(*

## Short summary
An interface to provide configurations for cycle manager steps.
Used internally to allow better fluent implementation.

.. <legal notes>

legal notes
=================
| SPDX-FileCopyrightText: © 2024 ekvip automation GmbH <info@ekvip.de>
| SPDX-License-Identifier: Apache-2.0
| For details check: Apache-2.0_

.. _Apache-2.0: https://www.apache.org/licenses/LICENSE-2.0

.. </legal notes>



*)
INTERFACE INTERNAL ICycleManagerStepParameters EXTENDS __System.IQueryInterface

PROPERTY currentErrorStep : DINT
SET
END_SET
END_PROPERTY

PROPERTY currentPauseEnabled : BOOL
SET
END_SET
END_PROPERTY

PROPERTY currentSteppingEnabled : BOOL
SET
END_SET
END_PROPERTY

PROPERTY currentStepWidth : DINT
SET
END_SET
END_PROPERTY

PROPERTY currentStopRequestMode :CNM_CycleManagerInterfaces.StepStopRequestMode
SET
END_SET
END_PROPERTY

PROPERTY currentTimeout : TIME
SET
END_SET
END_PROPERTY

PROPERTY currentTimeoutStep : DINT
SET
END_SET
END_PROPERTY

END_INTERFACE

(* stored: Version 1.1.0.1
   Itf ICycleManagerStepParameters: Id {5fd85db7-8dca-4b4c-bf21-26014628826b}
   Property currentErrorStep: Id {65d183e5-c0b6-4aea-b7a2-d27dc7ce9450}
   Set Set: Id {caa0b043-d1cd-423c-8f4d-f2bf68b0029e}
   Property currentPauseEnabled: Id {aed7e065-6f03-4e8b-88c8-55871102c280}
   Set Set: Id {270f9e99-f450-4f14-9a07-cce942922dfd}
   Property currentSteppingEnabled: Id {30211155-87f9-4899-bf47-99958d943402}
   Set Set: Id {711f4f81-8407-4fe4-a4af-e3076d0962c9}
   Property currentStepWidth: Id {5f8d236a-45af-4e6e-a44e-e4f099111d69}
   Set Set: Id {e59d0c31-506f-41d6-8815-fa0f3c2e4ccd}
   Property currentStopRequestMode: Id {264aa1b0-d87e-4301-ab6c-77034040f6ab}
   Set Set: Id {9fcdf647-e480-4225-be91-3725941f178e}
   Property currentTimeout: Id {ace83772-6f6b-4247-b50a-1841dba3ef52}
   Set Set: Id {ec393d65-b88f-4f92-8fa9-341ecfdfff33}
   Property currentTimeoutStep: Id {d9ca41eb-73dd-47e4-b5e4-673117fc2e76}
   Set Set: Id {5dac76aa-5be4-4954-83f9-8d430b54903e} *)
